RoboDK station: simple_ur5e_station.rdk

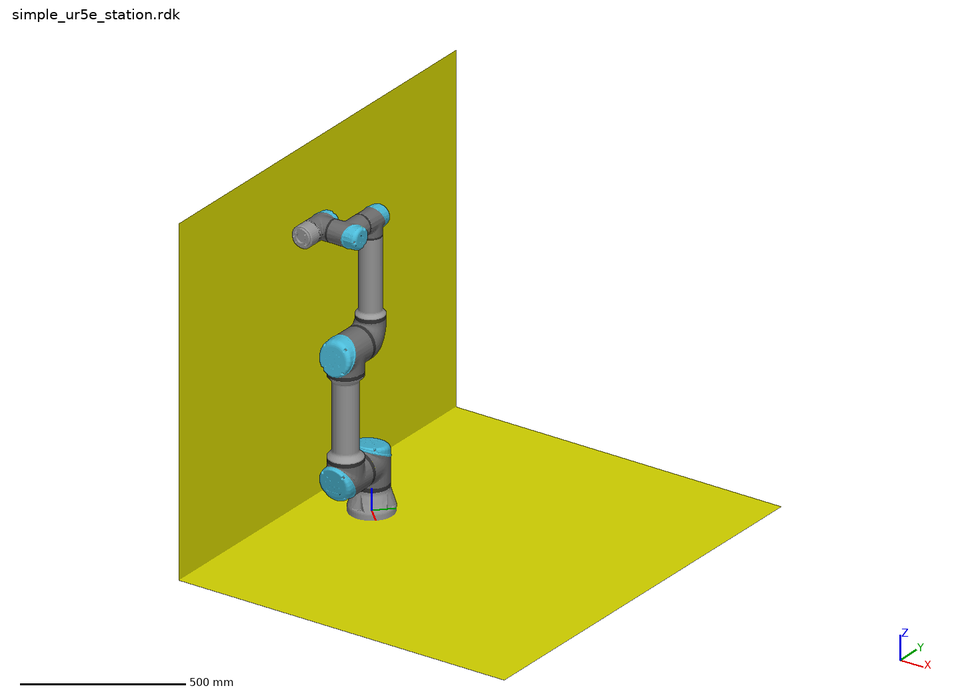
[picture v0: the station drawn from its stored meshes, robots at their saved joint values, targets as dots, program paths as lines]
Station simple_ur5e_station. Poses are relative to the parent item; angles as X-Y-Z fixed-axis rotations.
Station parameters (name, value as stored): CollisionFreePlanner, UR5e, CollisionFreePlanner-Rob UR5e
  - frame UR5e Base at (0, 0, 0) mm, rotated rx 0 ry 0 rz -45 deg
    - robot UR5e: 6 axes, payload 5 kg, reach 850 mm, repeatability 0.03 mm, weight 18.4 kg
        modified DH rows (alpha deg, a mm, theta deg, d mm): 0, 0, 0, 162.5; 90, 0, 180, 0; 0, 425, 0, 0; 0, 392.25, 0, 133.3; -90, 0, 0, 99.7; 90, 0, 180, 99.6
        joint limits [-360, -360, -360, -360, -360, -360] to [360, 360, 360, 360, 360, 360]; home [0, -90, -90, 0, 90, 0]; saved at [45, -90, 0, 0, 0, 0]
  - object Right wall at (0, 0, 0) mm, size 1200 x 1200 x 0.6 mm, geometry from plane_1m.sld
  - object Floor at (0, 0, 0) mm, size 1200 x 1460 x 0.6 mm
  - object Left wall at (0, 0, 0) mm, size 1200 x 1200 x 0.6 mm, geometry from plane_1m.sld
  - object Back wall at (0, 0, 0) mm, rotated rx 0 ry -90 rz 0 deg, size 1200 x 1460 x 0.6 mm
  - object Front wall at (0, 0, 0) mm, rotated rx 0 ry -90 rz 0 deg, size 1200 x 1460 x 0.6 mm
